//==================================================================================================
//							Beckhoff Automation Poland
//									2.11.2018
//	Zarzadzeni trybami pracy i komendami - Satate Machine
// 	v1.2	|| TC v 3.1.4022.25		|| - dodano Initialization 
// 	v1.1	|| TC v 3.1.4022.4		|| - Aktualizacja - dodano test Abort z HMI 
// 	v1.0	|| TC v 3.1.4022.4		|| - Pierwsza wersja
//==================================================================================================
PROGRAM P_ModeStateManager
VAR
	//	GVL_Machine - HMI handling
	bHMIModeRequest_Automatic			: BOOL;
	bHMIModeRequest_Manual				: BOOL;
	bHMIModeRequest_Maintenance			: BOOL;
	
	bHMICommandRequest_Run				: BOOL;
	bHMICommandRequest_Stop				: BOOL;
	bHMICommandRequest_Reset			: BOOL;
	bHMICommandRequest_Restart			: BOOL;
	bHMICommandRequest_Abort			: BOOL;
	// Rising edge detection
	rtButtonAutomatic					: R_TRIG;
	rtButtonManual						: R_TRIG;
	rtButtonMaintenance					: R_TRIG;
	rtButtonStart						: R_TRIG;
	rtButtonReset						: R_TRIG;
	rtButtonStop						: R_TRIG;
	// State change permissions
	bAllowChangeToManual				: BOOL;
	bAllowChangeToMaintenance			: BOOL;
	bAllowChangeToAutomatic				: BOOL;
END_VAR

// Triggers
rtButtonAutomatic(CLK:= bHMIModeRequest_Automatic);
rtButtonManual(CLK:= bHMIModeRequest_Manual);
rtButtonMaintenance(CLK:= bHMIModeRequest_Maintenance);
rtButtonStart(CLK:= GVL_IO.di_PBStart OR bHMICommandRequest_Run);
rtButtonStop(CLK:= GVL_IO.di_PBStop OR bHMICommandRequest_Stop);
rtButtonReset(CLK:= GVL_IO.di_PBReset OR bHMICommandRequest_Reset);

// SAFETY niezaleznie
IF NOT GVL_IO.bSAFETY_PermissionSS1 OR bHMICommandRequest_Abort THEN
	GVL_Machine.eCommand						:= E_MachineCommand.eAbort;
	GVL_Machine.eState							:= E_MachineState.eAborted;
END_IF
		
CASE GVL_Machine.eMode OF 

	E_MachineMode.eInitialization:

		// Reset just in case of init error
		P_Initialization(bReset := (P_Initialization.bError AND rtButtonReset.Q), bTestMode := );
		IF P_Initialization.bInitialized THEN
			// Choose mode to go
			GVL_Machine.eMode						:= E_MachineMode.eManual;
		END_IF
		
	E_MachineMode.eAutomatic:

		// Zmiana trybu tylko gdy maszyna nie jest w Running
		IF GVL_Machine.eState <> E_MachineState.eRunning THEN
			IF rtButtonMaintenance.Q THEN
				GVL_Machine.eState				:= E_MachineState.eIdle;
				GVL_Machine.eMode				:= E_MachineMode.eMaintenance;
			END_IF
		END_IF

		//==============================================
		IF rtButtonStart.Q THEN 
			GVL_Machine.eCommand 	:= E_MachineCommand.eRun;
		END_IF

		IF rtButtonReset.Q AND GVL.bRestartRequired THEN
			GVL_Machine.eCommand	:= E_MachineCommand.eRestart;
		END_IF
		
		IF rtButtonReset.Q AND NOT GVL.bRestartRequired THEN
			GVL_Machine.eCommand	:= E_MachineCommand.eReset;
		END_IF
		
		IF GVL.bGeneralError OR GVL.bGeneralFatalError OR rtButtonStop.Q THEN
			GVL_Machine.eCommand	:= E_MachineCommand.eStop ;
		END_IF
		
	E_MachineMode.eMaintenance, E_MachineMode.eManual:
	
		// Reset, Restart, Error - not used
		
		// Zmiana trybu tylko gdy maszyna nie jest w Running
		IF GVL_Machine.eState <> E_MachineState.eRunning THEN
			IF rtButtonAutomatic.Q (* OR sth *) THEN
				GVL_Machine.eState				:= E_MachineState.eIdle;
				GVL_Machine.eMode				:= E_MachineMode.eAutomatic;
			END_IF
		END_IF
		
		//==============================================
		IF rtButtonStart.Q THEN 
			GVL_Machine.eCommand 	:= E_MachineCommand.eRun;
		END_IF

		IF rtButtonReset.Q AND GVL.bRestartRequired THEN
			GVL_Machine.eCommand	:= E_MachineCommand.eRestart;
		END_IF
		
		IF rtButtonReset.Q AND NOT GVL.bRestartRequired THEN
			GVL_Machine.eCommand	:= E_MachineCommand.eReset;
		END_IF
		
		IF rtButtonStop.Q THEN
			GVL_Machine.eCommand	:= E_MachineCommand.eStop ;
		END_IF

END_CASE

ACTION Act_CollectMachineState:
// Action to decide global machine state
GVL_Machine.eState; // :=
END_ACTION

ACTION Act_ModeChangeSelector:
bAllowChangeToManual 				:= NOT (P_Template.eMachineState <> E_MachineState.eRunning); //
bAllowChangeToMaintenance;
bAllowChangeToAutomatic;
END_ACTION

END_PROGRAM

(* stored: Version 1.1.0.1, ProductVersion 3.1.4022.12
   POU P_ModeStateManager: Id {bbac15c0-b65a-450f-84c9-d78a3c906803}, SpecialFunc None
   Action Act_CollectMachineState: Id {35dbdadd-8e9d-4826-9020-b6db73a59fd4}
   Action Act_ModeChangeSelector: Id {93e687b8-71f2-4f96-a92e-dc8cc9cabd1b} *)
